ABB RobotStudio station: Task1_welding_DONE.rspag

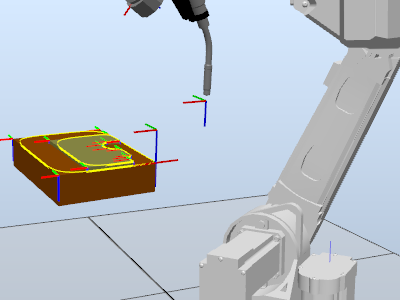
--- station ---
Station Task1_welding (saved by RobotStudio 22.2.10013.1)
Controller IRB_1520ID_4kg_1.50m
  mechanical unit ROB_1: IRB1520ID_4_150__02, 6 joints, base frame (0, 0, 0) mm
Layout (positions relative to the parent item):
  - IRB1520ID_4_150__02 [mechanism, from Robots\IRB1520ID_4_150_G_02.rslib] at (0, 0, 0) mm; joint values [0.6819, -0.4334, 0.4774, -0.8741, 1.9379, 2.0233] (rad or m)
  - AW_Gun_PSF_25 [mechanism, from Tools\AW_Gun_PSF_25.rslib] at (529.96, 245.81, 1039.9) mm, rotated rx 171.11 ry 53.87 rz 89.85 deg
  - Curve_thing [part, from Training Objects\Curve_Thing.rslib] at (696.55, 149.94, 458.64) mm, rotated rx 0 ry -5.23 rz 7.04 deg
Attachment: AW_Gun_PSF_25 is attached to IRB1520ID_4_150__02 / Link6
Targets, tools, work objects and paths stored in the station and not in the controller backup, written as RAPID:
! task T_ROB1
MODULE Module1
  PROC Path_10()
    MoveL Target_10,v1000,z100,AW_Gun\WObj:=Workobject_1;
    MoveL Target_20,v1000,z100,AW_Gun\WObj:=Workobject_1;
    MoveL Target_30,v1000,z100,AW_Gun\WObj:=Workobject_1;
    MoveL Target_40,v1000,z100,AW_Gun\WObj:=Workobject_1;
    MoveL Target_50,v1000,z100,AW_Gun\WObj:=Workobject_1;
  ENDPROC
  PROC Path_20()
    MoveL Target_60,v1000,z100,AW_Gun\WObj:=Workobject_1;
    MoveL Target_70,v1000,z100,AW_Gun\WObj:=Workobject_1;
    MoveL Target_80,v1000,z100,AW_Gun\WObj:=Workobject_1;
    MoveL Target_90,v1000,z100,AW_Gun\WObj:=Workobject_1;
    MoveL Target_100,v1000,z100,AW_Gun\WObj:=Workobject_1;
    MoveL Target_110,v1000,z100,AW_Gun\WObj:=Workobject_1;
    MoveL Target_120,v1000,z100,AW_Gun\WObj:=Workobject_1;
    MoveL Target_130,v1000,z100,AW_Gun\WObj:=Workobject_1;
    MoveL Target_140,v1000,z100,AW_Gun\WObj:=Workobject_1;
    MoveL Target_150,v1000,z100,AW_Gun\WObj:=Workobject_1;
    MoveL Target_160,v1000,z100,AW_Gun\WObj:=Workobject_1;
    MoveL Target_170,v1000,z100,AW_Gun\WObj:=Workobject_1;
    MoveL Target_180,v1000,z100,AW_Gun\WObj:=Workobject_1;
  ENDPROC
ENDMODULE


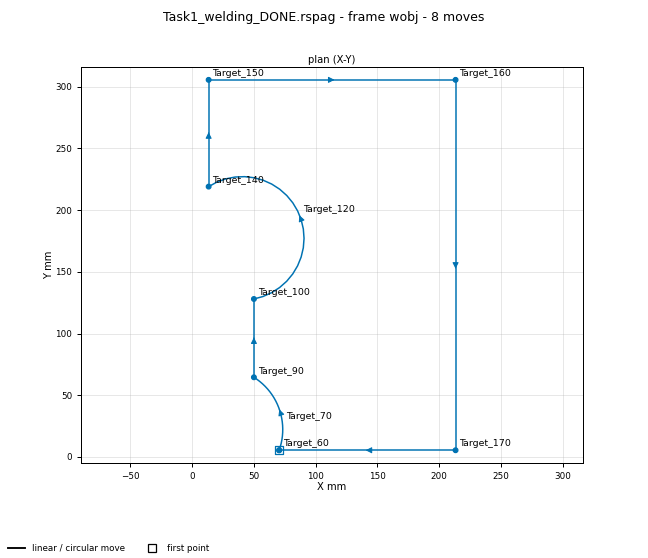
[picture p0: tool path of Task1_welding_DONE.rspag in frame wobj, 8 of 17 moves have a stored position in this frame; points joined in program order, loops and branches not executed]
--- Backups/IRB_1520ID_4kg_1.50m/RAPID/TASK1/PROGMOD/CalibData.mod ---
MODULE CalibData
	PERS tooldata AW_Gun:=[TRUE,[[119.5,0,352],[0.890213743,0,0.455543074,0]],[1,[0,0,100],[1,0,0,0],0,0,0]];
	TASK PERS wobjdata myPalletWO:=[FALSE,TRUE,"",[[688.418839009,148.925896983,548.269503166],[0.74843401,0.03415564,-0.030194721,-0.66164054]],[[0,0,0],[1,0,0,0]]];
    TASK PERS wobjdata Workobject_1:=[FALSE,TRUE,"",[[688.418,148.926,548.269],[0.030194646,0.661640544,0.748434013,0.034155555]],[[0,0,0],[1,0,0,0]]];
    TASK PERS wobjdata Workobject_2:=[FALSE,TRUE,"",[[679.378519985,147.808964582,647.853336283],[0.030194646,0.661640544,0.748434013,0.034155555]],[[0,0,0],[1,0,0,0]]];
ENDMODULE

--- Backups/IRB_1520ID_4kg_1.50m/RAPID/TASK1/PROGMOD/Module1.mod ---
MODULE Module1


    CONST robtarget Target_10:=[[-0.000424899,0.000383785,-0.000175989],[1,0,0,0],[0,0,0,0],[9E+09,9E+09,9E+09,9E+09,9E+09,9E+09]];
    CONST robtarget Target_20:=[[-0.000409879,400.000383785,-0.000515042],[1,0,0,0],[0,0,0,0],[9E+09,9E+09,9E+09,9E+09,9E+09,9E+09]];
    CONST robtarget Target_30:=[[299.999590121,400.000372519,-0.000516124],[1,-0.000000424,0.000000002,-0.000000019],[0,0,0,0],[9E+09,9E+09,9E+09,9E+09,9E+09,9E+09]];
    CONST robtarget Target_40:=[[299.9995751,0.00037252,-0.000177072],[1,0,0,0],[0,0,0,0],[9E+09,9E+09,9E+09,9E+09,9E+09,9E+09]];
    CONST robtarget Target_50:=[[-0.000424899,0.000383785,-0.000175989],[1,0,0,0],[0,0,0,0],[9E+09,9E+09,9E+09,9E+09,9E+09,9E+09]];
    CONST robtarget Target_60:=[[70.452202903,5.448141829,-10.000180861],[1,0,0,0],[0,0,0,0],[9E+09,9E+09,9E+09,9E+09,9E+09,9E+09]];
    CONST robtarget Target_70:=[[73.061891459,27.625951979,-10.00019967],[1,0,0,0],[0,0,0,0],[9E+09,9E+09,9E+09,9E+09,9E+09,9E+09]];
    CONST robtarget Target_80:=[[65.756453349,48.727997174,-10.00021753],[1,0,0,0],[0,0,0,0],[9E+09,9E+09,9E+09,9E+09,9E+09,9E+09]];
    CONST robtarget Target_90:=[[49.993077244,64.545130644,-10.000230881],[1,0,0,0],[0,0,0,0],[9E+09,9E+09,9E+09,9E+09,9E+09,9E+09]];
    CONST robtarget Target_100:=[[49.993079626,127.965328691,-10.000284637],[1,0,0,0],[0,0,0,0],[9E+09,9E+09,9E+09,9E+09,9E+09,9E+09]];
    CONST robtarget Target_110:=[[84.495149815,153.128794126,-10.000306091],[1,0,0,0],[0,0,0,0],[9E+09,9E+09,9E+09,9E+09,9E+09,9E+09]];
    CONST robtarget Target_120:=[[86.980415303,195.759959903,-10.000342236],[1,0,0,0],[0,0,0,0],[9E+09,9E+09,9E+09,9E+09,9E+09,9E+09]];
    CONST robtarget Target_130:=[[55.63603115,224.762070553,-10.000366706],[1,0,0,0],[0,0,0,0],[9E+09,9E+09,9E+09,9E+09,9E+09,9E+09]];
    CONST robtarget Target_140:=[[13.325755162,218.979909544,-10.000361652],[1,0,0,0],[0,0,0,0],[9E+09,9E+09,9E+09,9E+09,9E+09,9E+09]];
    CONST robtarget Target_150:=[[13.32575841,305.448143973,-10.000434944],[1,0,0,0],[0,0,0,0],[9E+09,9E+09,9E+09,9E+09,9E+09,9E+09]];
    CONST robtarget Target_160:=[[213.325758409,305.448136463,-10.000435666],[1,0,0,0],[0,0,0,0],[9E+09,9E+09,9E+09,9E+09,9E+09,9E+09]];
    CONST robtarget Target_170:=[[213.325747144,5.448136463,-10.000181377],[1,0,0,0],[0,0,0,0],[9E+09,9E+09,9E+09,9E+09,9E+09,9E+09]];
    CONST robtarget Target_180:=[[70.452202903,5.448141829,-10.000180861],[1,0,0,0],[0,0,0,0],[9E+09,9E+09,9E+09,9E+09,9E+09,9E+09]];


! Module:  Module1
    !
    ! Description:
    !   <Insert description here>
    !
    ! Author: Administrator
    !
    ! Version: 1.0
    !
    !***********************************************************


    !***********************************************************
    !
    ! Procedure main
    !
    !   This is the entry point of your program
    !
    !***********************************************************


    PROC main()

        Outer_profile 0;
        Inner_profile Workobject_1;
        MoveJ Offs(Target_10, -100,-100,-100), v800, z10,AW_Gun\WObj:=Workobject_1;
        WaitTime 3;
        ! can do like this
        Outer_profile 100;
        ! Or like this
        Inner_profile Workobject_2;
        MoveJ Offs(Target_10, -100,-100,-100), v800, z10,AW_Gun\WObj:=Workobject_2;
    ENDPROC

    PROC Inner_profile(PERS wobjdata wobj)

        VAR robtarget top_60;
        top_60:=Offs(Target_60,0,0,-50);
        ! this also possible for round shapes:
        MoveJ top_60, v1000,z0,AW_Gun\WObj:=wobj;
        MoveL Target_60,v1000,z0,AW_Gun\WObj:=wobj;
        MoveC Target_70, Target_90,v1000,z0,AW_Gun\WObj:=wobj;
        MoveL Target_100,v1000,z0,AW_Gun\WObj:=wobj;
        MoveC Target_120, Target_140,v1000,z0,AW_Gun\WObj:=wobj;
        MoveL Target_150,v1000,z0,AW_Gun\WObj:=wobj;
        MoveL Target_160,v1000,z0,AW_Gun\WObj:=wobj;
        MoveL Target_170,v1000,z0,AW_Gun\WObj:=wobj;
        MoveL Target_180,v1000,z0,AW_Gun\WObj:=wobj;
    ENDPROC

    PROC Outer_profile(num offsetinZ)
        !define targets for offsetting
        VAR robtarget top_10;
        VAR robtarget t_10;
        VAR robtarget t_20;
        VAR robtarget t_30;
        VAR robtarget t_40;
        VAR robtarget t_50;

        top_10:=Offs(Target_10,0,0,-100-offsetinZ);
        t_10:=Offs(Target_10,0,0,-offsetinZ);
        t_20:=Offs(Target_20,0,0,-offsetinZ);
        t_30:=Offs(Target_30,0,0,-offsetinZ);
        t_40:=Offs(Target_40,0,0,-offsetinZ);
        t_50:=Offs(Target_50,0,0,-offsetinZ);

        !movements
        MoveJ Top_10,v1000,z0,AW_Gun\WObj:=Workobject_1;
        MoveL t_10,v1000,z0,AW_Gun\WObj:=Workobject_1;
        MoveL t_20,v1000,z0,AW_Gun\WObj:=Workobject_1;
        MoveL t_30,v1000,z0,AW_Gun\WObj:=Workobject_1;
        MoveL t_40,v1000,z0,AW_Gun\WObj:=Workobject_1;
        MoveL t_50,v1000,z100,AW_Gun\WObj:=Workobject_1;
    ENDPROC


ENDMODULE

--- Backups/IRB_1520ID_4kg_1.50m/RAPID/TASK1/SYSMOD/LINKEDM.sys ---
%%%
  VERSION:1
  LANGUAGE:ENGLISH
%%%

MODULE LINKEDM (SYSMODULE)

! FOLLOWER
!     Name of electronically linked follower axis used by operator at teach pendent.
      PERS string l_f_axis_name{5}       :=  ["",  "", "", "", ""];

!     Name of the mechanical unit for follower axis.
      PERS string l_f_mecunt_n{5}  :=  ["", "", "", "", ""];

!     Linked follower axis number in the mechanical unit (first axis in mech. unit is number 1).
      PERS num l_f_axis_no{5}      :=  [0,          0,   0,  0,  0];

! MASTER
!     Name of the mechanical unit for linked master axis.
      PERS string l_m_mecunt_n{5} :=  ["", "", "", "", ""];

!     Linked master axis number in the mechanical unit (first axis in mech. unit is number 1).
!     See axis number table in documentation for different master mechanical units.
      PERS num l_m_axis_no{5}     :=  [0,  0,  0,  0,  0];

! POSITION OFFSET
!     The increase of the allowed offset position between the master and follower
!     positions, used when starting AUTO mode. As soon as the offset is decreased
!     the old configurated parameter is used.
!     Example: 3 => the configurated value of allowed offset is increased 3 times.
      PERS num offset_ratio{5}       :=  [10,  10,   10,  10,  10];

! SPEED RATIO
!     Speed_ratio used in AUTO and JOG modes [ very_slow   slow    normal    fast]
!     Value 1 = max allowed manual speed.
      CONST num speed_ratio {20}      := [0.01, 0.01, 0.01, 0.01, 0.01,
                                          0.05, 0.05, 0.05, 0.05, 0.05,
                                          0.20, 0.20, 0.20, 0.20, 0.20,
                                          1.00, 1.00, 1.00, 1.00, 1.00];

! STEP SIZE
!     Displacement position used in JOG mode for each activation of positive or
!     negative movement.                  [very_short    short   normal   long]
!     Unit degees or meter.
      CONST num displacement {20}     := [0.001, 0.001, 0.001, 0.001, 0.001,
                                          0.005, 0.005, 0.005, 0.005, 0.005,
                                          0.020, 0.020, 0.020, 0.020, 0.020,
                                          0.100, 0.100, 0.100, 0.100, 0.100];


!-------------------------------------------------------------
 PROC Linked_m ()
      Linked_m_exe ;
 ENDPROC
ENDMODULE
